DATA_BLOCK "dbArchiveParConveyor"
{ S7_Optimized_Access := 'TRUE' }
VERSION : 0.8
NON_RETAIN
"fbArchiveParConveyor"

BEGIN

END_DATA_BLOCK

